TYPE stResetHistory :
STRUCT
	sWorkerID					: STRING(255);
	sOperationDescription		: STRING(255);
	stDate						: stAircomTimeStruct;
	iOperationAmout				: ULINT;
	iCyclesAmount				: ULINT;
END_STRUCT
END_TYPE

(* stored: Version 1.1.0.1, ProductVersion 3.1.4024.13
   DUT stResetHistory: Id {ce57d3dc-c6ea-0f76-3f2f-e9d37760a9f1} *)
